// TwinCAT 3 PLC project PLC1
// ProgramVersion: 3.1.4024.0
// libraries:
//   SPT Base Types, * (Beckhoff Automation LLC)
//   Tc2_Standard, * (Beckhoff Automation GmbH)
//   Tc2_System, * (Beckhoff Automation GmbH)
//   Tc3_Module, * (Beckhoff Automation GmbH)
//   XPlanarApplication, * (Beckhoff Automation LLC)
// project tree:
//   / PlcTask.TcTTO
//   POUs/ MAIN.TcPOU
// real-time tasks:
//   TASK XPlanar Task3: cycle T#250us, priority 1, ADS port 350
//   TASK MC-Task (MET): cycle T#2ms, priority 2, ADS port 351
//   TASK MC-Task (MPT): cycle T#10ms, priority 3, ADS port 352
//   TASK Job Task: cycle default, priority 4
//   TASK PlcTask: cycle T#10ms, priority 20, ADS port 353
// variable links:
//   XPlanar MC Project/Axes/Mover4220_1 <-> TcCOM Objects/XPlanar/Mover4220_1
//     McToIo/STD <-> InputsFromNC3/NC3ToHW
//   PLC1/PLC1 Instance <-> XPlanar MC Project/Axes/Mover4220_1
//     PlcTask Inputs/MAIN.Mover._Mover.MCTOPLC/ACT <-> McToPlc/ACT
//     PlcTask Inputs/MAIN.Mover._Mover.MCTOPLC/COORDMODE <-> McToPlc/COORDMODE
//     PlcTask Inputs/MAIN.Mover._Mover.MCTOPLC/SET <-> McToPlc/SET
//     PlcTask Inputs/MAIN.Mover._Mover.MCTOPLC/SETONTRACK <-> McToPlc/SETONTRACK
//     PlcTask Inputs/MAIN.Mover._Mover.MCTOPLC/STD <-> McToPlc/STD
//     PlcTask Outputs/MAIN.Mover._Mover.PLCTOMC/STD <-> PlcToMc/STD
//   PLC1/PLC1 Instance <-> XPlanar MC Project/Groups/Environment
//     PlcTask Inputs/XPlanarApplication.XPlanar.Environment.MCTOPLC_STD <-> McToPlc/STD
//   PLC1/PLC1 Instance <-> XPlanar MC Project/Groups/XPlanar
//     PlcTask Inputs/XPlanarApplication.XPlanar.Group.MCTOPLC_STD <-> McToPlc/STD
//   TcCOM Objects/XPlanar/Mover4220_1 <-> XPlanar MC Project/Axes/Mover4220_1
//     OutputsToNC3/HWToNC3 <-> IoToMc/STD

CONFIGURATION PLC1
    RESOURCE PLC ON TwinCAT3
        TASK PlcTask(INTERVAL := T#10ms, PRIORITY := 20);
        PROGRAM MAIN WITH PlcTask : MAIN;
    END_RESOURCE
END_CONFIGURATION

// ---- POUs/MAIN.TcPOU
PROGRAM MAIN
VAR
	XPlanarTable  : FB_Component_XPlanar;
	Mover		  : FB_XPlanarMover;
	i			  : UDINT;
	EnableMovers  : BOOL;
	DisableMovers : BOOL;
	MoveCmd1	  : BOOL;
	MoveCmd2	  : BOOL;
	CommandResult : I_PlanarTaskResult;
END_VAR

//Set the intefaces for background functions **This must be done first!**
ip.Movers[1] := Mover;

//Keep the XPlanar System up to date
XplanarTable.CyclicLogic();

//Enable movers
IF EnableMovers THEN
	IF Mover.Enable().Done THEN
		EnableMovers := FALSE; 
	END_IF
END_IF

//DisableMovers
IF DisableMovers THEN
	IF Mover.Disable().Done THEN
		DisableMovers := FALSE;
	END_IF
END_IF

//Move 1
IF MoveCmd1 THEN
	IF Mover.MoveCommand.FreeMove(120, 360).Done THEN
		MoveCmd1 := FALSE;
	END_IF
END_IF

//Move 2
IF MoveCmd2 THEN
	IF Mover.MoveCommand.FreeMove(120, 120).Done THEN
		MoveCmd2 := FALSE;
	END_IF	
END_IF

END_PROGRAM
